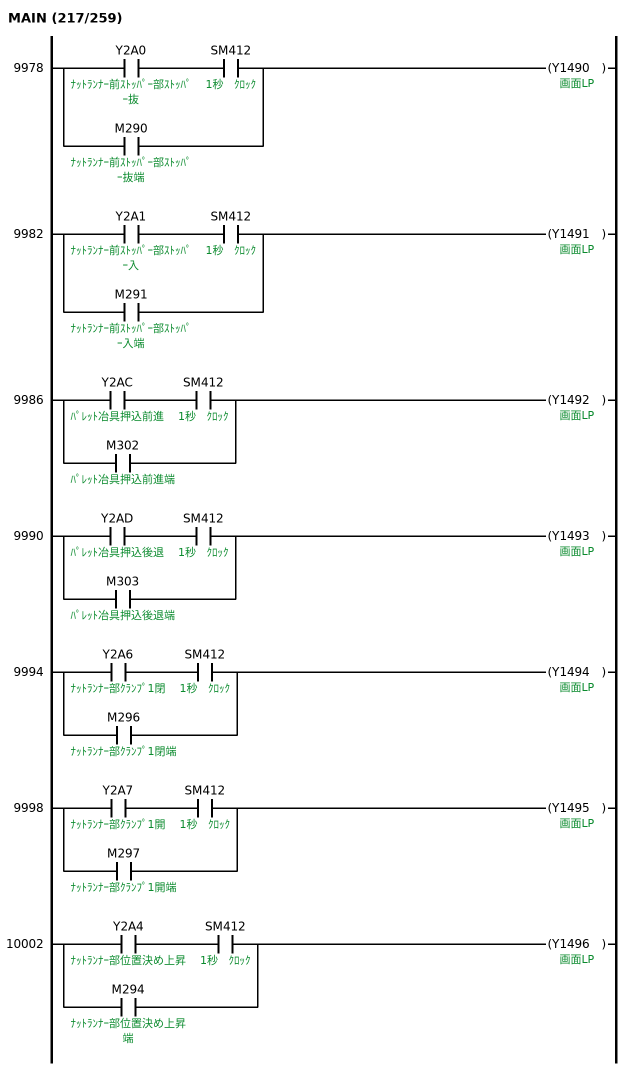
[picture p216: ladder of MAIN, rungs at steps 9978 to 10002]
9978  LD      Y2A0  ; ﾅｯﾄﾗﾝﾅｰ前ｽﾄｯﾊﾟｰ部ｽﾄｯﾊﾟｰ抜
      AND     SM412  ; 1秒   ｸﾛｯｸ
      OR      M290  ; ﾅｯﾄﾗﾝﾅｰ前ｽﾄｯﾊﾟｰ部ｽﾄｯﾊﾟｰ抜端
      OUT     Y1490  ; 画面LP
9982  LD      Y2A1  ; ﾅｯﾄﾗﾝﾅｰ前ｽﾄｯﾊﾟｰ部ｽﾄｯﾊﾟｰ入
      AND     SM412  ; 1秒   ｸﾛｯｸ
      OR      M291  ; ﾅｯﾄﾗﾝﾅｰ前ｽﾄｯﾊﾟｰ部ｽﾄｯﾊﾟｰ入端
      OUT     Y1491  ; 画面LP
9986  LD      Y2AC  ; ﾊﾟﾚｯﾄ冶具押込前進
      AND     SM412  ; 1秒   ｸﾛｯｸ
      OR      M302  ; ﾊﾟﾚｯﾄ冶具押込前進端
      OUT     Y1492  ; 画面LP
9990  LD      Y2AD  ; ﾊﾟﾚｯﾄ冶具押込後退
      AND     SM412  ; 1秒   ｸﾛｯｸ
      OR      M303  ; ﾊﾟﾚｯﾄ冶具押込後退端
      OUT     Y1493  ; 画面LP
9994  LD      Y2A6  ; ﾅｯﾄﾗﾝﾅｰ部ｸﾗﾝﾌﾟ1閉
      AND     SM412  ; 1秒   ｸﾛｯｸ
      OR      M296  ; ﾅｯﾄﾗﾝﾅｰ部ｸﾗﾝﾌﾟ1閉端
      OUT     Y1494  ; 画面LP
9998  LD      Y2A7  ; ﾅｯﾄﾗﾝﾅｰ部ｸﾗﾝﾌﾟ1開
      AND     SM412  ; 1秒   ｸﾛｯｸ
      OR      M297  ; ﾅｯﾄﾗﾝﾅｰ部ｸﾗﾝﾌﾟ1開端
      OUT     Y1495  ; 画面LP
10002 LD      Y2A4  ; ﾅｯﾄﾗﾝﾅｰ部位置決め上昇
      AND     SM412  ; 1秒   ｸﾛｯｸ
      OR      M294  ; ﾅｯﾄﾗﾝﾅｰ部位置決め上昇端
      OUT     Y1496  ; 画面LP
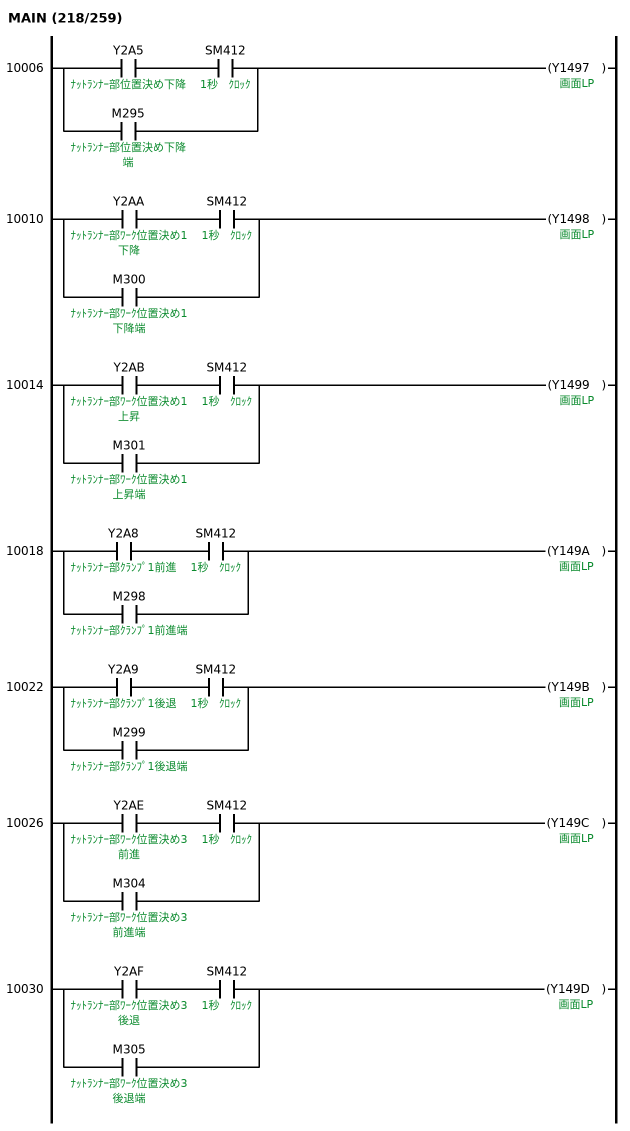
10006 LD      Y2A5  ; ﾅｯﾄﾗﾝﾅｰ部位置決め下降
      AND     SM412  ; 1秒   ｸﾛｯｸ
      OR      M295  ; ﾅｯﾄﾗﾝﾅｰ部位置決め下降端
      OUT     Y1497  ; 画面LP
10010 LD      Y2AA  ; ﾅｯﾄﾗﾝﾅｰ部ﾜｰｸ位置決め1下降
      AND     SM412  ; 1秒   ｸﾛｯｸ
      OR      M300  ; ﾅｯﾄﾗﾝﾅｰ部ﾜｰｸ位置決め1下降端
      OUT     Y1498  ; 画面LP
10014 LD      Y2AB  ; ﾅｯﾄﾗﾝﾅｰ部ﾜｰｸ位置決め1上昇
      AND     SM412  ; 1秒   ｸﾛｯｸ
      OR      M301  ; ﾅｯﾄﾗﾝﾅｰ部ﾜｰｸ位置決め1上昇端
      OUT     Y1499  ; 画面LP
10018 LD      Y2A8  ; ﾅｯﾄﾗﾝﾅｰ部ｸﾗﾝﾌﾟ1前進
      AND     SM412  ; 1秒   ｸﾛｯｸ
      OR      M298  ; ﾅｯﾄﾗﾝﾅｰ部ｸﾗﾝﾌﾟ1前進端
      OUT     Y149A  ; 画面LP
10022 LD      Y2A9  ; ﾅｯﾄﾗﾝﾅｰ部ｸﾗﾝﾌﾟ1後退
      AND     SM412  ; 1秒   ｸﾛｯｸ
      OR      M299  ; ﾅｯﾄﾗﾝﾅｰ部ｸﾗﾝﾌﾟ1後退端
      OUT     Y149B  ; 画面LP
10026 LD      Y2AE  ; ﾅｯﾄﾗﾝﾅｰ部ﾜｰｸ位置決め3前進
      AND     SM412  ; 1秒   ｸﾛｯｸ
      OR      M304  ; ﾅｯﾄﾗﾝﾅｰ部ﾜｰｸ位置決め3前進端
      OUT     Y149C  ; 画面LP
10030 LD      Y2AF  ; ﾅｯﾄﾗﾝﾅｰ部ﾜｰｸ位置決め3後退
      AND     SM412  ; 1秒   ｸﾛｯｸ
      OR      M305  ; ﾅｯﾄﾗﾝﾅｰ部ﾜｰｸ位置決め3後退端
      OUT     Y149D  ; 画面LP
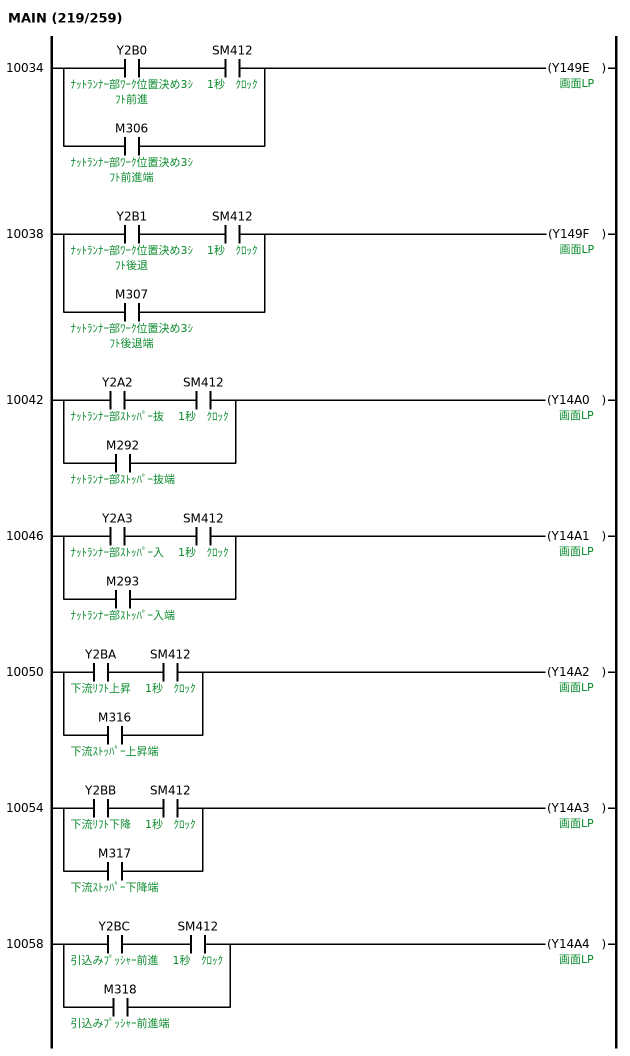
10034 LD      Y2B0  ; ﾅｯﾄﾗﾝﾅｰ部ﾜｰｸ位置決め3ｼﾌﾄ前進
      AND     SM412  ; 1秒   ｸﾛｯｸ
      OR      M306  ; ﾅｯﾄﾗﾝﾅｰ部ﾜｰｸ位置決め3ｼﾌﾄ前進端
      OUT     Y149E  ; 画面LP
10038 LD      Y2B1  ; ﾅｯﾄﾗﾝﾅｰ部ﾜｰｸ位置決め3ｼﾌﾄ後退
      AND     SM412  ; 1秒   ｸﾛｯｸ
      OR      M307  ; ﾅｯﾄﾗﾝﾅｰ部ﾜｰｸ位置決め3ｼﾌﾄ後退端
      OUT     Y149F  ; 画面LP
10042 LD      Y2A2  ; ﾅｯﾄﾗﾝﾅｰ部ｽﾄｯﾊﾟｰ抜
      AND     SM412  ; 1秒   ｸﾛｯｸ
      OR      M292  ; ﾅｯﾄﾗﾝﾅｰ部ｽﾄｯﾊﾟｰ抜端
      OUT     Y14A0  ; 画面LP
10046 LD      Y2A3  ; ﾅｯﾄﾗﾝﾅｰ部ｽﾄｯﾊﾟｰ入
      AND     SM412  ; 1秒   ｸﾛｯｸ
      OR      M293  ; ﾅｯﾄﾗﾝﾅｰ部ｽﾄｯﾊﾟｰ入端
      OUT     Y14A1  ; 画面LP
10050 LD      Y2BA  ; 下流ﾘﾌﾄ上昇
      AND     SM412  ; 1秒   ｸﾛｯｸ
      OR      M316  ; 下流ｽﾄｯﾊﾟｰ上昇端
      OUT     Y14A2  ; 画面LP
10054 LD      Y2BB  ; 下流ﾘﾌﾄ下降
      AND     SM412  ; 1秒   ｸﾛｯｸ
      OR      M317  ; 下流ｽﾄｯﾊﾟｰ下降端
      OUT     Y14A3  ; 画面LP
10058 LD      Y2BC  ; 引込みﾌﾟｯｼｬｰ前進
      AND     SM412  ; 1秒   ｸﾛｯｸ
      OR      M318  ; 引込みﾌﾟｯｼｬｰ前進端
      OUT     Y14A4  ; 画面LP
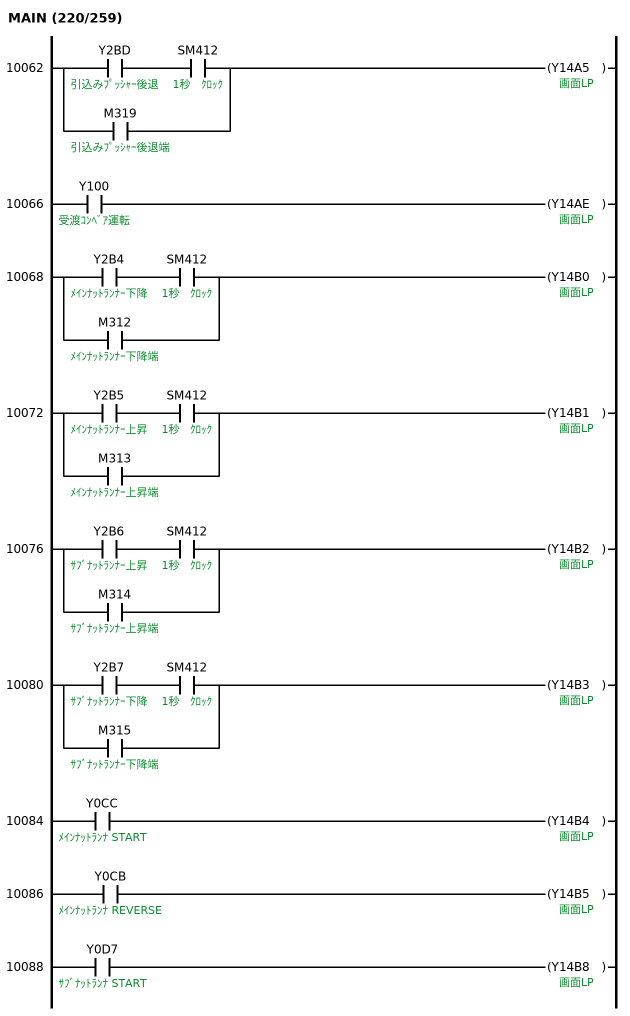
10062 LD      Y2BD  ; 引込みﾌﾟｯｼｬｰ後退
      AND     SM412  ; 1秒   ｸﾛｯｸ
      OR      M319  ; 引込みﾌﾟｯｼｬｰ後退端
      OUT     Y14A5  ; 画面LP
10066 LD      Y100  ; 受渡ｺﾝﾍﾞｱ運転
      OUT     Y14AE  ; 画面LP
10068 LD      Y2B4  ; ﾒｲﾝﾅｯﾄﾗﾝﾅｰ下降
      AND     SM412  ; 1秒   ｸﾛｯｸ
      OR      M312  ; ﾒｲﾝﾅｯﾄﾗﾝﾅｰ下降端
      OUT     Y14B0  ; 画面LP
10072 LD      Y2B5  ; ﾒｲﾝﾅｯﾄﾗﾝﾅｰ上昇
      AND     SM412  ; 1秒   ｸﾛｯｸ
      OR      M313  ; ﾒｲﾝﾅｯﾄﾗﾝﾅｰ上昇端
      OUT     Y14B1  ; 画面LP
10076 LD      Y2B6  ; ｻﾌﾞﾅｯﾄﾗﾝﾅｰ上昇
      AND     SM412  ; 1秒   ｸﾛｯｸ
      OR      M314  ; ｻﾌﾞﾅｯﾄﾗﾝﾅｰ上昇端
      OUT     Y14B2  ; 画面LP
10080 LD      Y2B7  ; ｻﾌﾞﾅｯﾄﾗﾝﾅｰ下降
      AND     SM412  ; 1秒   ｸﾛｯｸ
      OR      M315  ; ｻﾌﾞﾅｯﾄﾗﾝﾅｰ下降端
      OUT     Y14B3  ; 画面LP
10084 LD      Y0CC  ; ﾒｲﾝﾅｯﾄﾗﾝﾅ START
      OUT     Y14B4  ; 画面LP
10086 LD      Y0CB  ; ﾒｲﾝﾅｯﾄﾗﾝﾅ REVERSE
      OUT     Y14B5  ; 画面LP
10088 LD      Y0D7  ; ｻﾌﾞﾅｯﾄﾗﾝﾅ START
      OUT     Y14B8  ; 画面LP
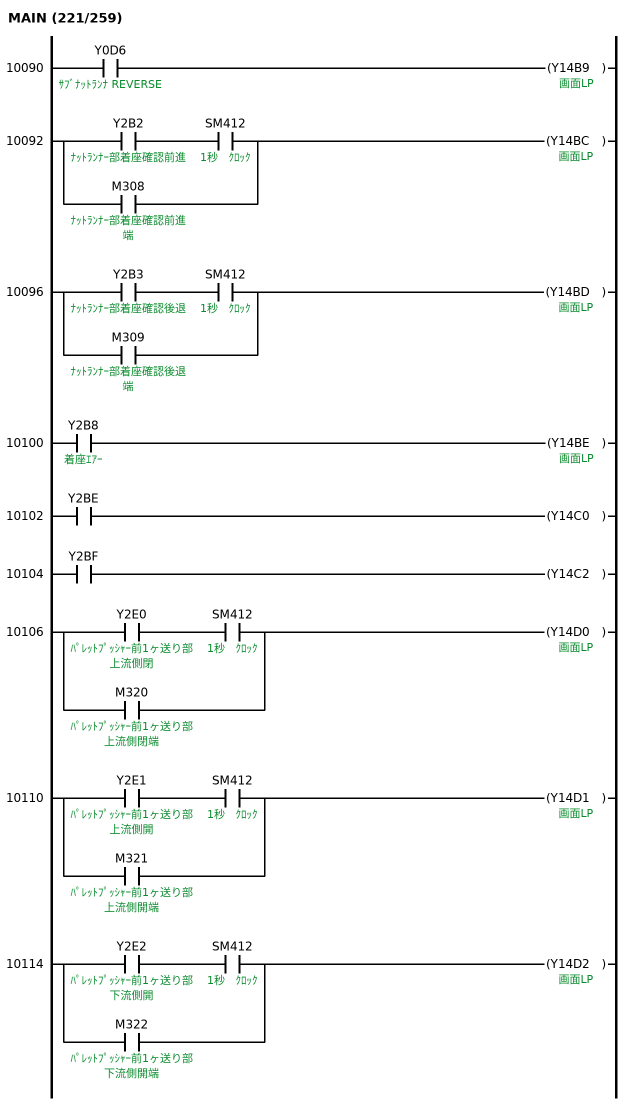
10090 LD      Y0D6  ; ｻﾌﾞﾅｯﾄﾗﾝﾅ REVERSE
      OUT     Y14B9  ; 画面LP
10092 LD      Y2B2  ; ﾅｯﾄﾗﾝﾅｰ部着座確認前進
      AND     SM412  ; 1秒   ｸﾛｯｸ
      OR      M308  ; ﾅｯﾄﾗﾝﾅｰ部着座確認前進端
      OUT     Y14BC  ; 画面LP
10096 LD      Y2B3  ; ﾅｯﾄﾗﾝﾅｰ部着座確認後退
      AND     SM412  ; 1秒   ｸﾛｯｸ
      OR      M309  ; ﾅｯﾄﾗﾝﾅｰ部着座確認後退端
      OUT     Y14BD  ; 画面LP
10100 LD      Y2B8  ; 着座ｴｱｰ
      OUT     Y14BE  ; 画面LP
10102 LD      Y2BE
      OUT     Y14C0
10104 LD      Y2BF
      OUT     Y14C2
10106 LD      Y2E0  ; ﾊﾟﾚｯﾄﾌﾟｯｼｬｰ前1ヶ送り部上流側閉
      AND     SM412  ; 1秒   ｸﾛｯｸ
      OR      M320  ; ﾊﾟﾚｯﾄﾌﾟｯｼｬｰ前1ヶ送り部上流側閉端
      OUT     Y14D0  ; 画面LP
10110 LD      Y2E1  ; ﾊﾟﾚｯﾄﾌﾟｯｼｬｰ前1ヶ送り部上流側開
      AND     SM412  ; 1秒   ｸﾛｯｸ
      OR      M321  ; ﾊﾟﾚｯﾄﾌﾟｯｼｬｰ前1ヶ送り部上流側開端
      OUT     Y14D1  ; 画面LP
10114 LD      Y2E2  ; ﾊﾟﾚｯﾄﾌﾟｯｼｬｰ前1ヶ送り部下流側開
      AND     SM412  ; 1秒   ｸﾛｯｸ
      OR      M322  ; ﾊﾟﾚｯﾄﾌﾟｯｼｬｰ前1ヶ送り部下流側開端
      OUT     Y14D2  ; 画面LP
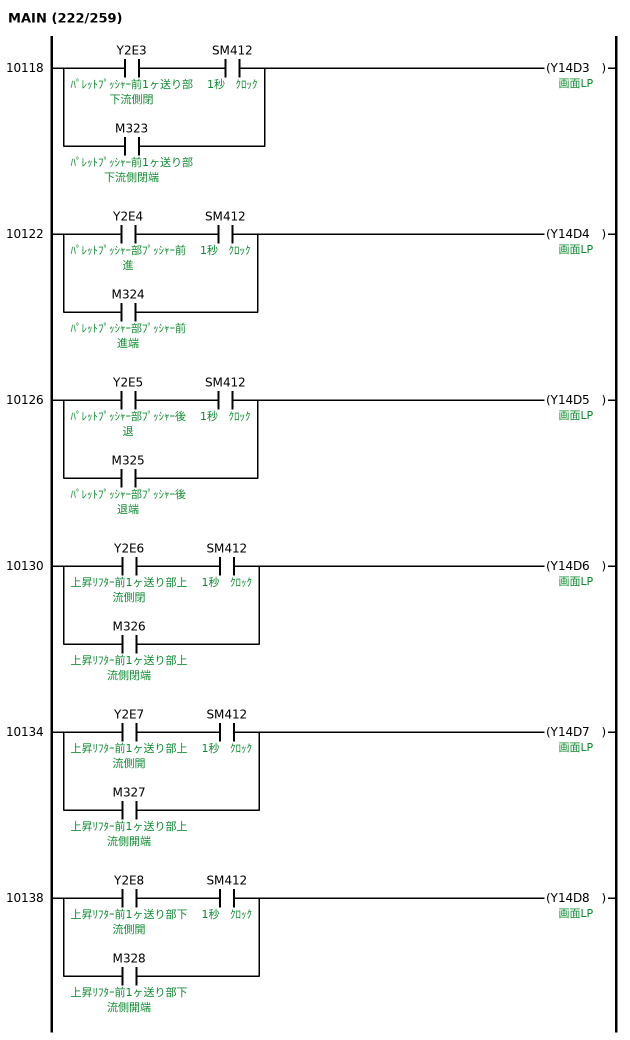
10118 LD      Y2E3  ; ﾊﾟﾚｯﾄﾌﾟｯｼｬｰ前1ヶ送り部下流側閉
      AND     SM412  ; 1秒   ｸﾛｯｸ
      OR      M323  ; ﾊﾟﾚｯﾄﾌﾟｯｼｬｰ前1ヶ送り部下流側閉端
      OUT     Y14D3  ; 画面LP
10122 LD      Y2E4  ; ﾊﾟﾚｯﾄﾌﾟｯｼｬｰ部ﾌﾟｯｼｬｰ前進
      AND     SM412  ; 1秒   ｸﾛｯｸ
      OR      M324  ; ﾊﾟﾚｯﾄﾌﾟｯｼｬｰ部ﾌﾟｯｼｬｰ前進端
      OUT     Y14D4  ; 画面LP
10126 LD      Y2E5  ; ﾊﾟﾚｯﾄﾌﾟｯｼｬｰ部ﾌﾟｯｼｬｰ後退
      AND     SM412  ; 1秒   ｸﾛｯｸ
      OR      M325  ; ﾊﾟﾚｯﾄﾌﾟｯｼｬｰ部ﾌﾟｯｼｬｰ後退端
      OUT     Y14D5  ; 画面LP
10130 LD      Y2E6  ; 上昇ﾘﾌﾀｰ前1ヶ送り部上流側閉
      AND     SM412  ; 1秒   ｸﾛｯｸ
      OR      M326  ; 上昇ﾘﾌﾀｰ前1ヶ送り部上流側閉端
      OUT     Y14D6  ; 画面LP
10134 LD      Y2E7  ; 上昇ﾘﾌﾀｰ前1ヶ送り部上流側開
      AND     SM412  ; 1秒   ｸﾛｯｸ
      OR      M327  ; 上昇ﾘﾌﾀｰ前1ヶ送り部上流側開端
      OUT     Y14D7  ; 画面LP
10138 LD      Y2E8  ; 上昇ﾘﾌﾀｰ前1ヶ送り部下流側開
      AND     SM412  ; 1秒   ｸﾛｯｸ
      OR      M328  ; 上昇ﾘﾌﾀｰ前1ヶ送り部下流側開端
      OUT     Y14D8  ; 画面LP
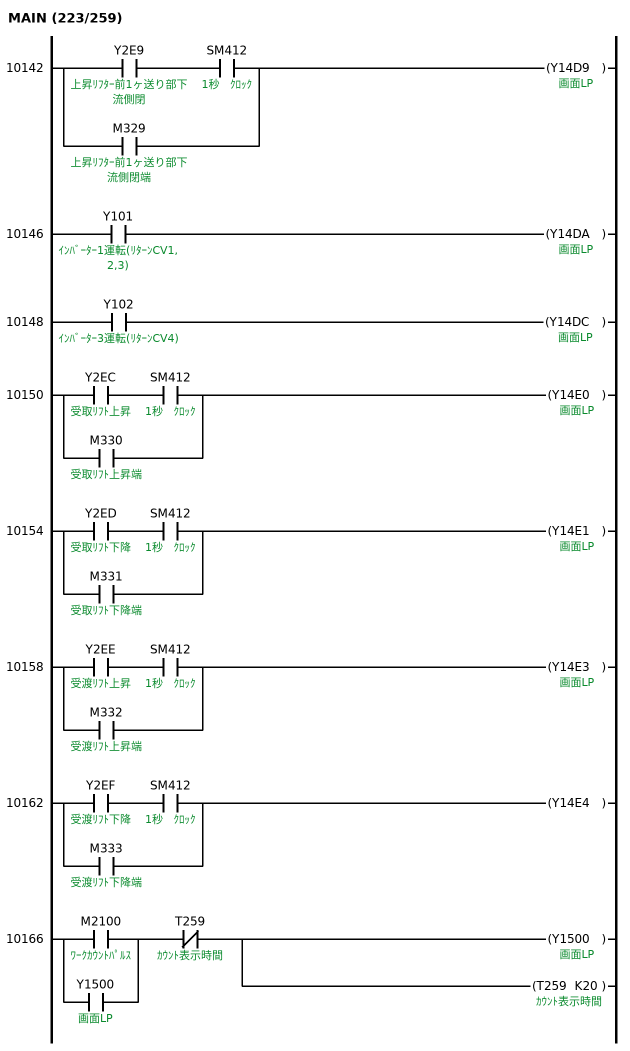
10142 LD      Y2E9  ; 上昇ﾘﾌﾀｰ前1ヶ送り部下流側閉
      AND     SM412  ; 1秒   ｸﾛｯｸ
      OR      M329  ; 上昇ﾘﾌﾀｰ前1ヶ送り部下流側閉端
      OUT     Y14D9  ; 画面LP
10146 LD      Y101  ; ｲﾝﾊﾞｰﾀｰ1運転(ﾘﾀｰﾝCV1,2,3)
      OUT     Y14DA  ; 画面LP
10148 LD      Y102  ; ｲﾝﾊﾞｰﾀｰ3運転(ﾘﾀｰﾝCV4)
      OUT     Y14DC  ; 画面LP
10150 LD      Y2EC  ; 受取ﾘﾌﾄ上昇
      AND     SM412  ; 1秒   ｸﾛｯｸ
      OR      M330  ; 受取ﾘﾌﾄ上昇端
      OUT     Y14E0  ; 画面LP
10154 LD      Y2ED  ; 受取ﾘﾌﾄ下降
      AND     SM412  ; 1秒   ｸﾛｯｸ
      OR      M331  ; 受取ﾘﾌﾄ下降端
      OUT     Y14E1  ; 画面LP
10158 LD      Y2EE  ; 受渡ﾘﾌﾄ上昇
      AND     SM412  ; 1秒   ｸﾛｯｸ
      OR      M332  ; 受渡ﾘﾌﾄ上昇端
      OUT     Y14E3  ; 画面LP
10162 LD      Y2EF  ; 受渡ﾘﾌﾄ下降
      AND     SM412  ; 1秒   ｸﾛｯｸ
      OR      M333  ; 受渡ﾘﾌﾄ下降端
      OUT     Y14E4
10166 LD      M2100  ; ﾜｰｸｶｳﾝﾄﾊﾟﾙｽ
      OR      Y1500  ; 画面LP
      ANI     T259  ; ｶｳﾝﾄ表示時間
      OUT     Y1500  ; 画面LP
      OUT     T259 K20  ; ｶｳﾝﾄ表示時間
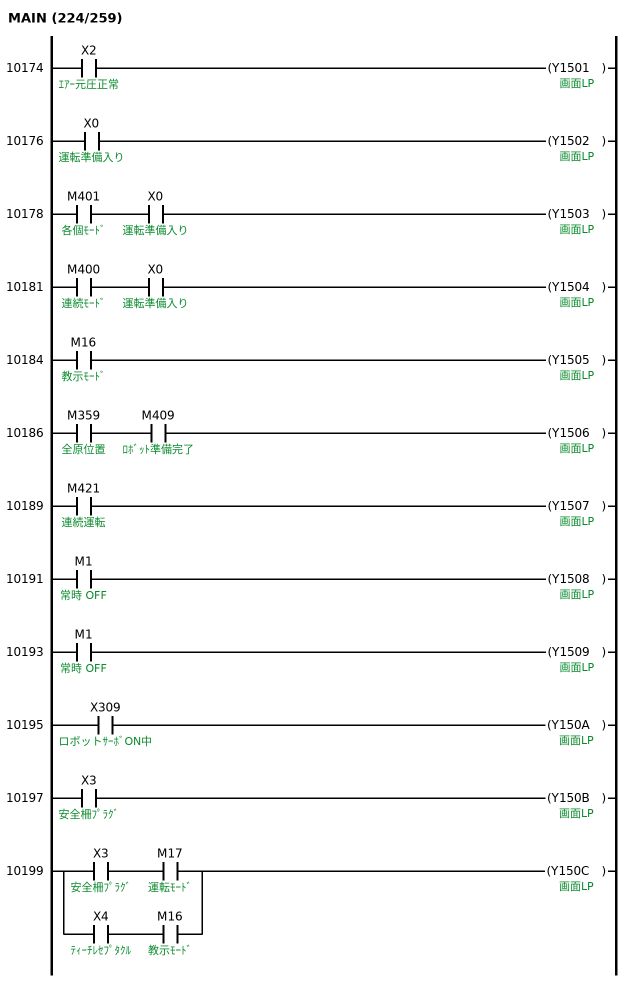
10174 LD      X2  ; ｴｱｰ元圧正常
      OUT     Y1501  ; 画面LP
10176 LD      X0  ; 運転準備入り
      OUT     Y1502  ; 画面LP
10178 LD      M401  ; 各個ﾓｰﾄﾞ
      AND     X0  ; 運転準備入り
      OUT     Y1503  ; 画面LP
10181 LD      M400  ; 連続ﾓｰﾄﾞ
      AND     X0  ; 運転準備入り
      OUT     Y1504  ; 画面LP
10184 LD      M16  ; 教示ﾓｰﾄﾞ
      OUT     Y1505  ; 画面LP
10186 LD      M359  ; 全原位置
      AND     M409  ; ﾛﾎﾞｯﾄ準備完了
      OUT     Y1506  ; 画面LP
10189 LD      M421  ; 連続運転
      OUT     Y1507  ; 画面LP
10191 LD      M1  ; 常時 OFF
      OUT     Y1508  ; 画面LP
10193 LD      M1  ; 常時 OFF
      OUT     Y1509  ; 画面LP
10195 LD      X309  ; ロボットｻｰﾎﾞON中
      OUT     Y150A  ; 画面LP
10197 LD      X3  ; 安全柵ﾌﾟﾗｸﾞ
      OUT     Y150B  ; 画面LP
10199 LD      X3  ; 安全柵ﾌﾟﾗｸﾞ
      AND     M17  ; 運転ﾓｰﾄﾞ
      LD      X4  ; ﾃｨｰﾁﾚｾﾌﾟﾀｸﾙ
      AND     M16  ; 教示ﾓｰﾄﾞ
      ORB
      OUT     Y150C  ; 画面LP
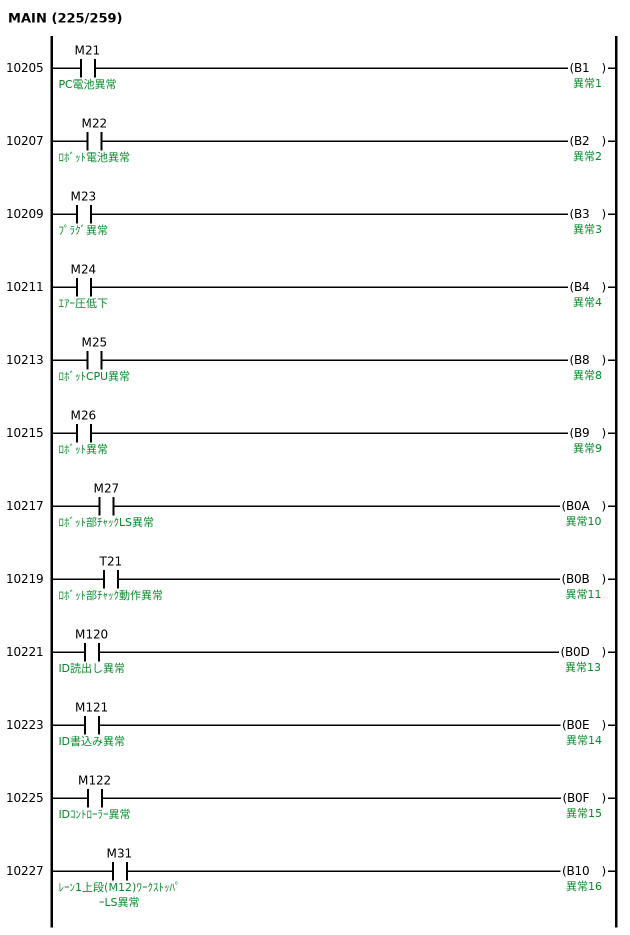
10205 LD      M21  ; PC電池異常
      OUT     B1  ; 異常1
10207 LD      M22  ; ﾛﾎﾞｯﾄ電池異常
      OUT     B2  ; 異常2
10209 LD      M23  ; ﾌﾟﾗｸﾞ異常
      OUT     B3  ; 異常3
10211 LD      M24  ; ｴｱｰ圧低下
      OUT     B4  ; 異常4
10213 LD      M25  ; ﾛﾎﾞｯﾄCPU異常
      OUT     B8  ; 異常8
10215 LD      M26  ; ﾛﾎﾞｯﾄ異常
      OUT     B9  ; 異常9
10217 LD      M27  ; ﾛﾎﾞｯﾄ部ﾁｬｯｸLS異常
      OUT     B0A  ; 異常10
10219 LD      T21  ; ﾛﾎﾞｯﾄ部ﾁｬｯｸ動作異常
      OUT     B0B  ; 異常11
10221 LD      M120  ; ID読出し異常
      OUT     B0D  ; 異常13
10223 LD      M121  ; ID書込み異常
      OUT     B0E  ; 異常14
10225 LD      M122  ; IDｺﾝﾄﾛｰﾗｰ異常
      OUT     B0F  ; 異常15
10227 LD      M31  ; ﾚｰﾝ1上段(M12)ﾜｰｸｽﾄｯﾊﾟｰLS異常
      OUT     B10  ; 異常16
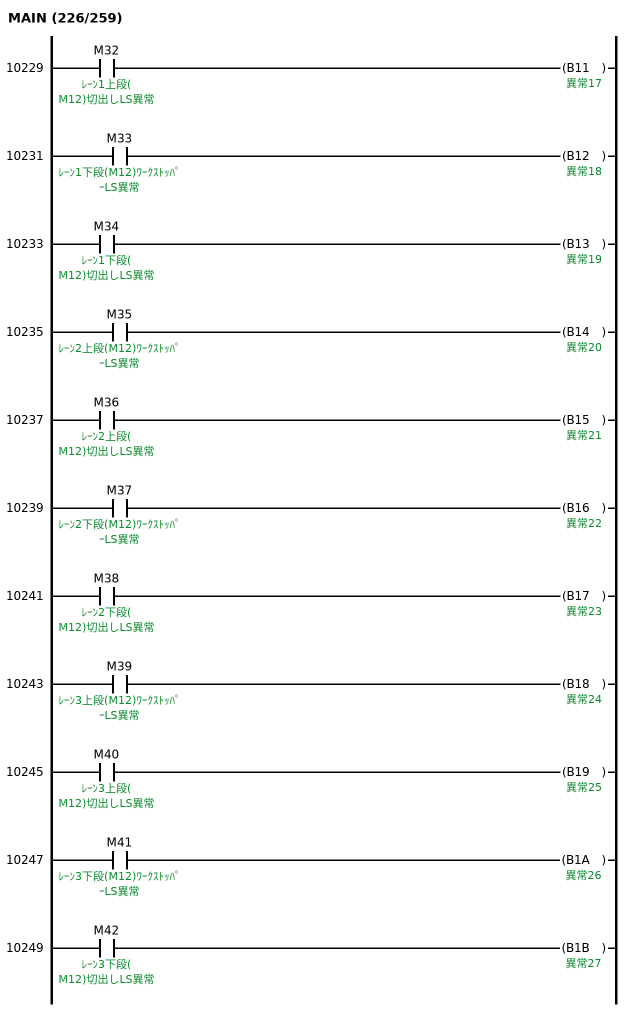
10229 LD      M32  ; ﾚｰﾝ1上段(M12)切出しLS異常
      OUT     B11  ; 異常17
10231 LD      M33  ; ﾚｰﾝ1下段(M12)ﾜｰｸｽﾄｯﾊﾟｰLS異常
      OUT     B12  ; 異常18
10233 LD      M34  ; ﾚｰﾝ1下段(M12)切出しLS異常
      OUT     B13  ; 異常19
10235 LD      M35  ; ﾚｰﾝ2上段(M12)ﾜｰｸｽﾄｯﾊﾟｰLS異常
      OUT     B14  ; 異常20
10237 LD      M36  ; ﾚｰﾝ2上段(M12)切出しLS異常
      OUT     B15  ; 異常21
10239 LD      M37  ; ﾚｰﾝ2下段(M12)ﾜｰｸｽﾄｯﾊﾟｰLS異常
      OUT     B16  ; 異常22
10241 LD      M38  ; ﾚｰﾝ2下段(M12)切出しLS異常
      OUT     B17  ; 異常23
10243 LD      M39  ; ﾚｰﾝ3上段(M12)ﾜｰｸｽﾄｯﾊﾟｰLS異常
      OUT     B18  ; 異常24
10245 LD      M40  ; ﾚｰﾝ3上段(M12)切出しLS異常
      OUT     B19  ; 異常25
10247 LD      M41  ; ﾚｰﾝ3下段(M12)ﾜｰｸｽﾄｯﾊﾟｰLS異常
      OUT     B1A  ; 異常26
10249 LD      M42  ; ﾚｰﾝ3下段(M12)切出しLS異常
      OUT     B1B  ; 異常27
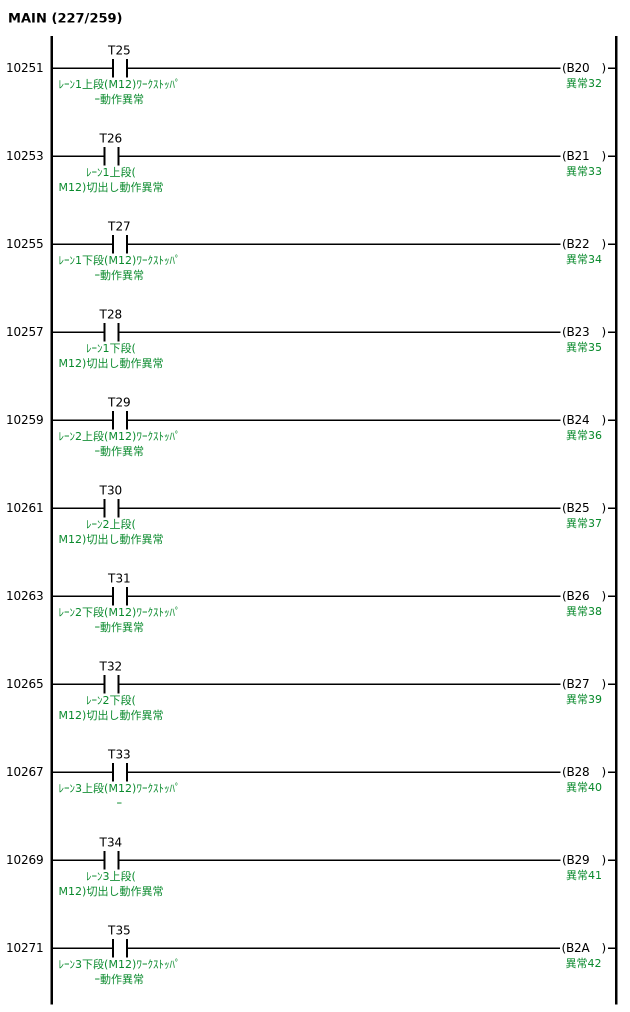
10251 LD      T25  ; ﾚｰﾝ1上段(M12)ﾜｰｸｽﾄｯﾊﾟｰ動作異常
      OUT     B20  ; 異常32
10253 LD      T26  ; ﾚｰﾝ1上段(M12)切出し動作異常
      OUT     B21  ; 異常33
10255 LD      T27  ; ﾚｰﾝ1下段(M12)ﾜｰｸｽﾄｯﾊﾟｰ動作異常
      OUT     B22  ; 異常34
10257 LD      T28  ; ﾚｰﾝ1下段(M12)切出し動作異常
      OUT     B23  ; 異常35
10259 LD      T29  ; ﾚｰﾝ2上段(M12)ﾜｰｸｽﾄｯﾊﾟｰ動作異常
      OUT     B24  ; 異常36
10261 LD      T30  ; ﾚｰﾝ2上段(M12)切出し動作異常
      OUT     B25  ; 異常37
10263 LD      T31  ; ﾚｰﾝ2下段(M12)ﾜｰｸｽﾄｯﾊﾟｰ動作異常
      OUT     B26  ; 異常38
10265 LD      T32  ; ﾚｰﾝ2下段(M12)切出し動作異常
      OUT     B27  ; 異常39
10267 LD      T33  ; ﾚｰﾝ3上段(M12)ﾜｰｸｽﾄｯﾊﾟｰ
      OUT     B28  ; 異常40
10269 LD      T34  ; ﾚｰﾝ3上段(M12)切出し動作異常
      OUT     B29  ; 異常41
10271 LD      T35  ; ﾚｰﾝ3下段(M12)ﾜｰｸｽﾄｯﾊﾟｰ動作異常
      OUT     B2A  ; 異常42
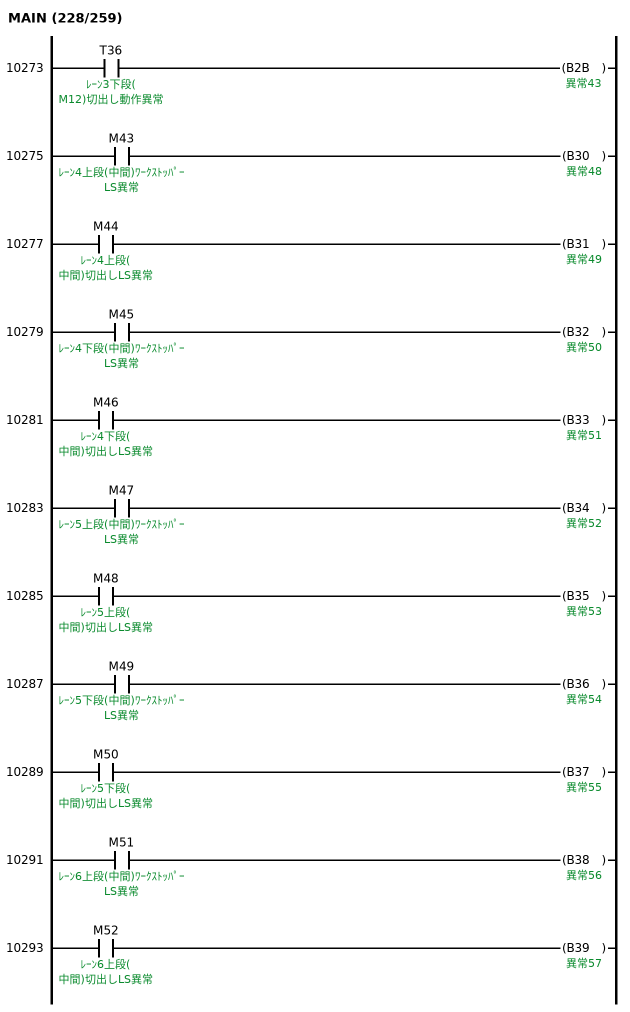
10273 LD      T36  ; ﾚｰﾝ3下段(M12)切出し動作異常
      OUT     B2B  ; 異常43
10275 LD      M43  ; ﾚｰﾝ4上段(中間)ﾜｰｸｽﾄｯﾊﾟｰLS異常
      OUT     B30  ; 異常48
10277 LD      M44  ; ﾚｰﾝ4上段(中間)切出しLS異常
      OUT     B31  ; 異常49
10279 LD      M45  ; ﾚｰﾝ4下段(中間)ﾜｰｸｽﾄｯﾊﾟｰLS異常
      OUT     B32  ; 異常50
10281 LD      M46  ; ﾚｰﾝ4下段(中間)切出しLS異常
      OUT     B33  ; 異常51
10283 LD      M47  ; ﾚｰﾝ5上段(中間)ﾜｰｸｽﾄｯﾊﾟｰLS異常
      OUT     B34  ; 異常52
10285 LD      M48  ; ﾚｰﾝ5上段(中間)切出しLS異常
      OUT     B35  ; 異常53
10287 LD      M49  ; ﾚｰﾝ5下段(中間)ﾜｰｸｽﾄｯﾊﾟｰLS異常
      OUT     B36  ; 異常54
10289 LD      M50  ; ﾚｰﾝ5下段(中間)切出しLS異常
      OUT     B37  ; 異常55
10291 LD      M51  ; ﾚｰﾝ6上段(中間)ﾜｰｸｽﾄｯﾊﾟｰLS異常
      OUT     B38  ; 異常56
10293 LD      M52  ; ﾚｰﾝ6上段(中間)切出しLS異常
      OUT     B39  ; 異常57
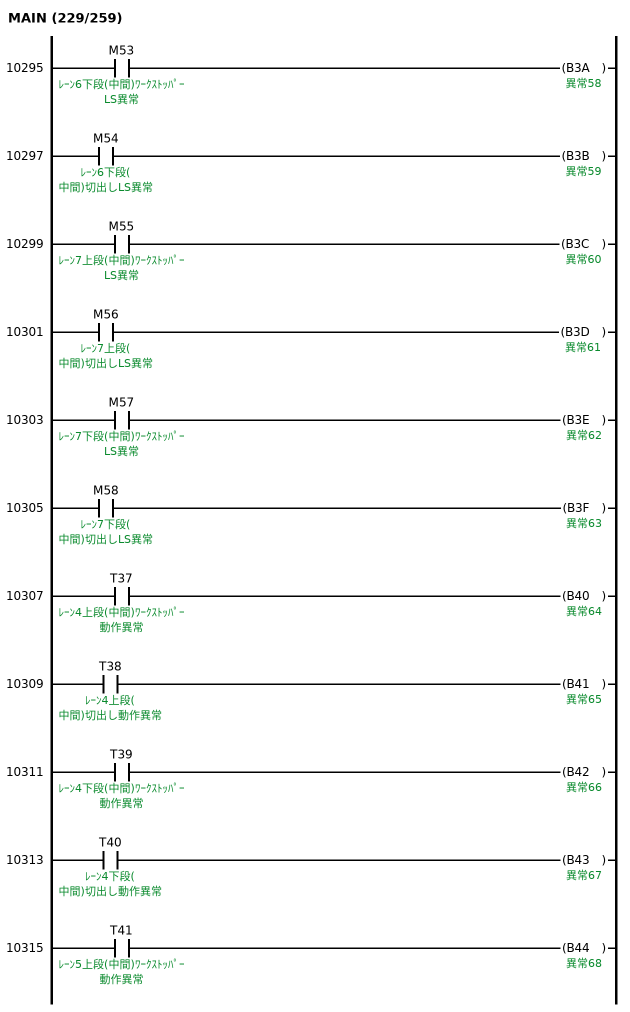
10295 LD      M53  ; ﾚｰﾝ6下段(中間)ﾜｰｸｽﾄｯﾊﾟｰLS異常
      OUT     B3A  ; 異常58
10297 LD      M54  ; ﾚｰﾝ6下段(中間)切出しLS異常
      OUT     B3B  ; 異常59
10299 LD      M55  ; ﾚｰﾝ7上段(中間)ﾜｰｸｽﾄｯﾊﾟｰLS異常
      OUT     B3C  ; 異常60
10301 LD      M56  ; ﾚｰﾝ7上段(中間)切出しLS異常
      OUT     B3D  ; 異常61
10303 LD      M57  ; ﾚｰﾝ7下段(中間)ﾜｰｸｽﾄｯﾊﾟｰLS異常
      OUT     B3E  ; 異常62
10305 LD      M58  ; ﾚｰﾝ7下段(中間)切出しLS異常
      OUT     B3F  ; 異常63
10307 LD      T37  ; ﾚｰﾝ4上段(中間)ﾜｰｸｽﾄｯﾊﾟｰ動作異常
      OUT     B40  ; 異常64
10309 LD      T38  ; ﾚｰﾝ4上段(中間)切出し動作異常
      OUT     B41  ; 異常65
10311 LD      T39  ; ﾚｰﾝ4下段(中間)ﾜｰｸｽﾄｯﾊﾟｰ動作異常
      OUT     B42  ; 異常66
10313 LD      T40  ; ﾚｰﾝ4下段(中間)切出し動作異常
      OUT     B43  ; 異常67
10315 LD      T41  ; ﾚｰﾝ5上段(中間)ﾜｰｸｽﾄｯﾊﾟｰ動作異常
      OUT     B44  ; 異常68
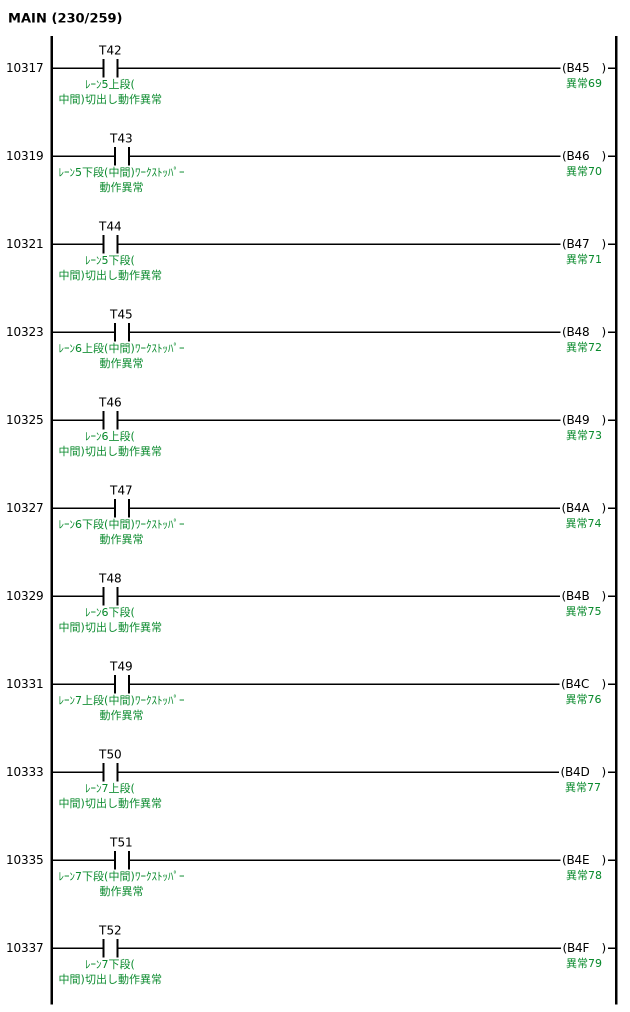
10317 LD      T42  ; ﾚｰﾝ5上段(中間)切出し動作異常
      OUT     B45  ; 異常69
10319 LD      T43  ; ﾚｰﾝ5下段(中間)ﾜｰｸｽﾄｯﾊﾟｰ動作異常
      OUT     B46  ; 異常70
10321 LD      T44  ; ﾚｰﾝ5下段(中間)切出し動作異常
      OUT     B47  ; 異常71
10323 LD      T45  ; ﾚｰﾝ6上段(中間)ﾜｰｸｽﾄｯﾊﾟｰ動作異常
      OUT     B48  ; 異常72
10325 LD      T46  ; ﾚｰﾝ6上段(中間)切出し動作異常
      OUT     B49  ; 異常73
10327 LD      T47  ; ﾚｰﾝ6下段(中間)ﾜｰｸｽﾄｯﾊﾟｰ動作異常
      OUT     B4A  ; 異常74
10329 LD      T48  ; ﾚｰﾝ6下段(中間)切出し動作異常
      OUT     B4B  ; 異常75
10331 LD      T49  ; ﾚｰﾝ7上段(中間)ﾜｰｸｽﾄｯﾊﾟｰ動作異常
      OUT     B4C  ; 異常76
10333 LD      T50  ; ﾚｰﾝ7上段(中間)切出し動作異常
      OUT     B4D  ; 異常77
10335 LD      T51  ; ﾚｰﾝ7下段(中間)ﾜｰｸｽﾄｯﾊﾟｰ動作異常
      OUT     B4E  ; 異常78
10337 LD      T52  ; ﾚｰﾝ7下段(中間)切出し動作異常
      OUT     B4F  ; 異常79
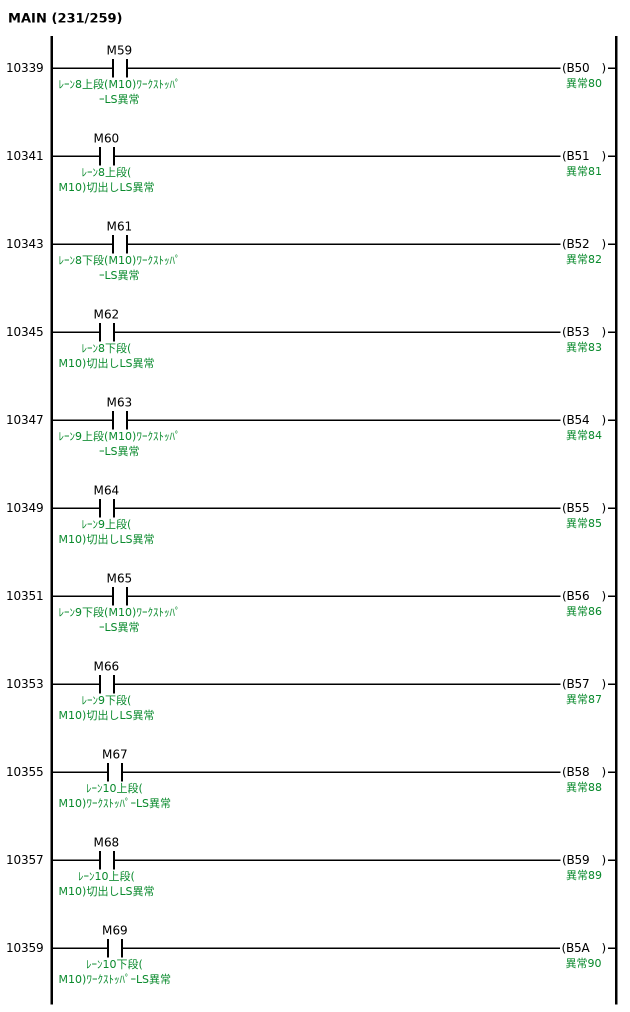
10339 LD      M59  ; ﾚｰﾝ8上段(M10)ﾜｰｸｽﾄｯﾊﾟｰLS異常
      OUT     B50  ; 異常80
10341 LD      M60  ; ﾚｰﾝ8上段(M10)切出しLS異常
      OUT     B51  ; 異常81
10343 LD      M61  ; ﾚｰﾝ8下段(M10)ﾜｰｸｽﾄｯﾊﾟｰLS異常
      OUT     B52  ; 異常82
10345 LD      M62  ; ﾚｰﾝ8下段(M10)切出しLS異常
      OUT     B53  ; 異常83
10347 LD      M63  ; ﾚｰﾝ9上段(M10)ﾜｰｸｽﾄｯﾊﾟｰLS異常
      OUT     B54  ; 異常84
10349 LD      M64  ; ﾚｰﾝ9上段(M10)切出しLS異常
      OUT     B55  ; 異常85
10351 LD      M65  ; ﾚｰﾝ9下段(M10)ﾜｰｸｽﾄｯﾊﾟｰLS異常
      OUT     B56  ; 異常86
10353 LD      M66  ; ﾚｰﾝ9下段(M10)切出しLS異常
      OUT     B57  ; 異常87
10355 LD      M67  ; ﾚｰﾝ10上段(M10)ﾜｰｸｽﾄｯﾊﾟｰLS異常
      OUT     B58  ; 異常88
10357 LD      M68  ; ﾚｰﾝ10上段(M10)切出しLS異常
      OUT     B59  ; 異常89
10359 LD      M69  ; ﾚｰﾝ10下段(M10)ﾜｰｸｽﾄｯﾊﾟｰLS異常
      OUT     B5A  ; 異常90
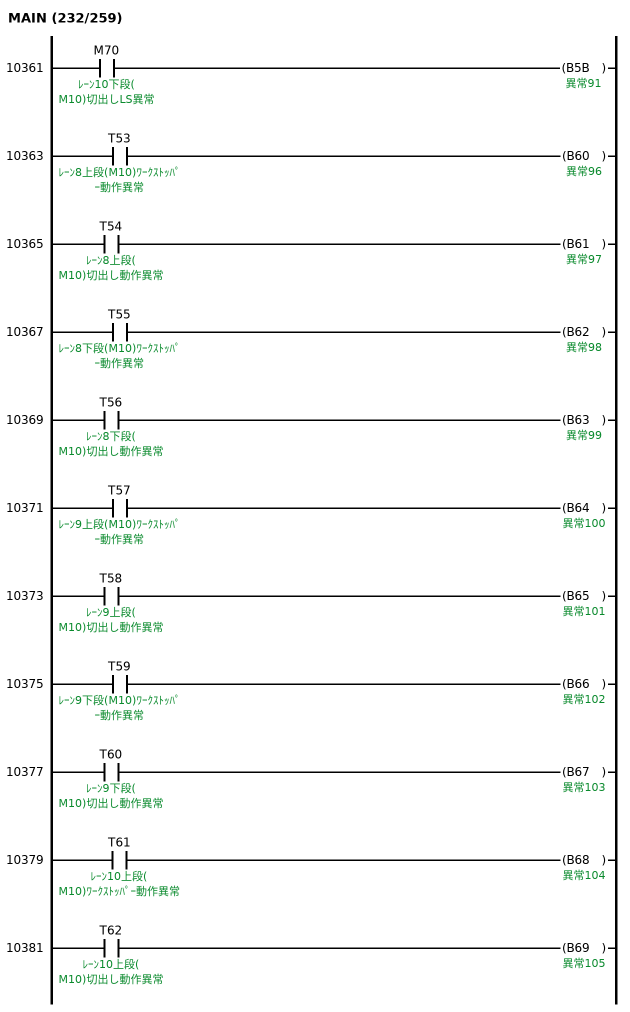
10361 LD      M70  ; ﾚｰﾝ10下段(M10)切出しLS異常
      OUT     B5B  ; 異常91
10363 LD      T53  ; ﾚｰﾝ8上段(M10)ﾜｰｸｽﾄｯﾊﾟｰ動作異常
      OUT     B60  ; 異常96
10365 LD      T54  ; ﾚｰﾝ8上段(M10)切出し動作異常
      OUT     B61  ; 異常97
10367 LD      T55  ; ﾚｰﾝ8下段(M10)ﾜｰｸｽﾄｯﾊﾟｰ動作異常
      OUT     B62  ; 異常98
10369 LD      T56  ; ﾚｰﾝ8下段(M10)切出し動作異常
      OUT     B63  ; 異常99
10371 LD      T57  ; ﾚｰﾝ9上段(M10)ﾜｰｸｽﾄｯﾊﾟｰ動作異常
      OUT     B64  ; 異常100
10373 LD      T58  ; ﾚｰﾝ9上段(M10)切出し動作異常
      OUT     B65  ; 異常101
10375 LD      T59  ; ﾚｰﾝ9下段(M10)ﾜｰｸｽﾄｯﾊﾟｰ動作異常
      OUT     B66  ; 異常102
10377 LD      T60  ; ﾚｰﾝ9下段(M10)切出し動作異常
      OUT     B67  ; 異常103
10379 LD      T61  ; ﾚｰﾝ10上段(M10)ﾜｰｸｽﾄｯﾊﾟｰ動作異常
      OUT     B68  ; 異常104
10381 LD      T62  ; ﾚｰﾝ10上段(M10)切出し動作異常
      OUT     B69  ; 異常105
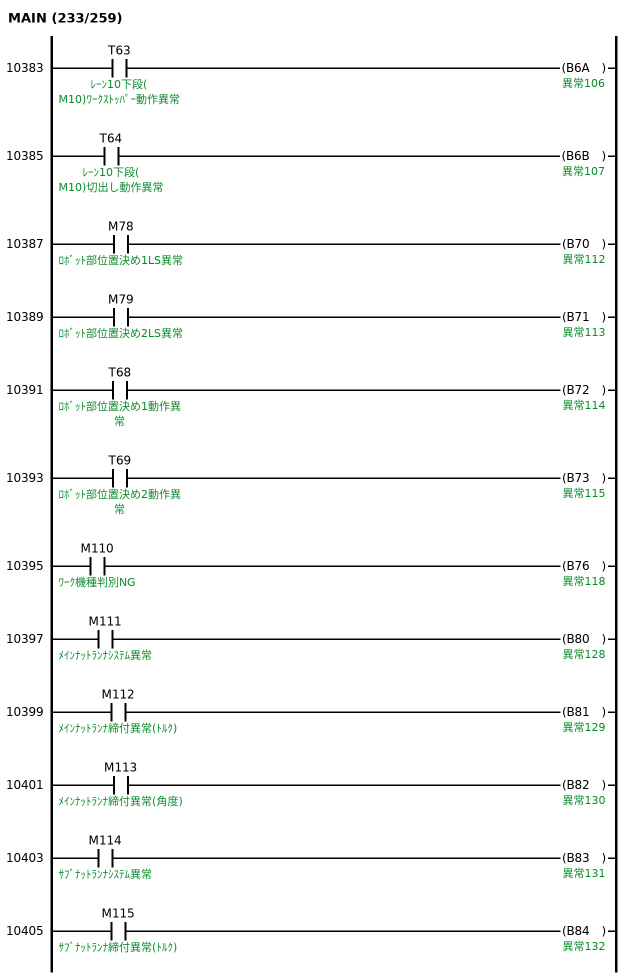
10383 LD      T63  ; ﾚｰﾝ10下段(M10)ﾜｰｸｽﾄｯﾊﾟｰ動作異常
      OUT     B6A  ; 異常106
10385 LD      T64  ; ﾚｰﾝ10下段(M10)切出し動作異常
      OUT     B6B  ; 異常107
10387 LD      M78  ; ﾛﾎﾞｯﾄ部位置決め1LS異常
      OUT     B70  ; 異常112
10389 LD      M79  ; ﾛﾎﾞｯﾄ部位置決め2LS異常
      OUT     B71  ; 異常113
10391 LD      T68  ; ﾛﾎﾞｯﾄ部位置決め1動作異常
      OUT     B72  ; 異常114
10393 LD      T69  ; ﾛﾎﾞｯﾄ部位置決め2動作異常
      OUT     B73  ; 異常115
10395 LD      M110  ; ﾜｰｸ機種判別NG
      OUT     B76  ; 異常118
10397 LD      M111  ; ﾒｲﾝﾅｯﾄﾗﾝﾅｼｽﾃﾑ異常
      OUT     B80  ; 異常128
10399 LD      M112  ; ﾒｲﾝﾅｯﾄﾗﾝﾅ締付異常(ﾄﾙｸ)
      OUT     B81  ; 異常129
10401 LD      M113  ; ﾒｲﾝﾅｯﾄﾗﾝﾅ締付異常(角度)
      OUT     B82  ; 異常130
10403 LD      M114  ; ｻﾌﾞﾅｯﾄﾗﾝﾅｼｽﾃﾑ異常
      OUT     B83  ; 異常131
10405 LD      M115  ; ｻﾌﾞﾅｯﾄﾗﾝﾅ締付異常(ﾄﾙｸ)
      OUT     B84  ; 異常132
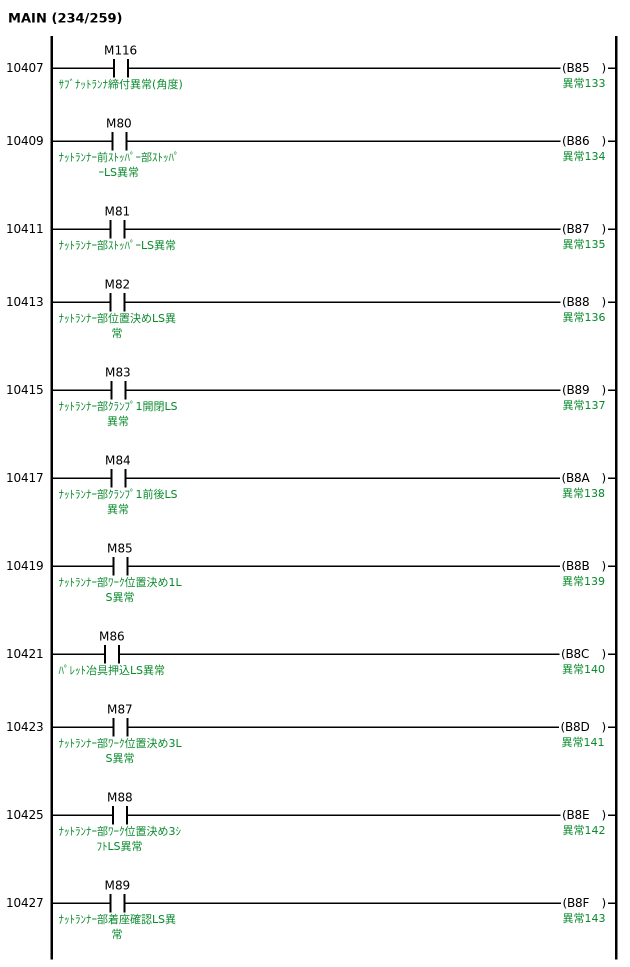
10407 LD      M116  ; ｻﾌﾞﾅｯﾄﾗﾝﾅ締付異常(角度)
      OUT     B85  ; 異常133
10409 LD      M80  ; ﾅｯﾄﾗﾝﾅｰ前ｽﾄｯﾊﾟｰ部ｽﾄｯﾊﾟｰLS異常
      OUT     B86  ; 異常134
10411 LD      M81  ; ﾅｯﾄﾗﾝﾅｰ部ｽﾄｯﾊﾟｰLS異常
      OUT     B87  ; 異常135
10413 LD      M82  ; ﾅｯﾄﾗﾝﾅｰ部位置決めLS異常
      OUT     B88  ; 異常136
10415 LD      M83  ; ﾅｯﾄﾗﾝﾅｰ部ｸﾗﾝﾌﾟ1開閉LS異常
      OUT     B89  ; 異常137
10417 LD      M84  ; ﾅｯﾄﾗﾝﾅｰ部ｸﾗﾝﾌﾟ1前後LS異常
      OUT     B8A  ; 異常138
10419 LD      M85  ; ﾅｯﾄﾗﾝﾅｰ部ﾜｰｸ位置決め1LS異常
      OUT     B8B  ; 異常139
10421 LD      M86  ; ﾊﾟﾚｯﾄ冶具押込LS異常
      OUT     B8C  ; 異常140
10423 LD      M87  ; ﾅｯﾄﾗﾝﾅｰ部ﾜｰｸ位置決め3LS異常
      OUT     B8D  ; 異常141
10425 LD      M88  ; ﾅｯﾄﾗﾝﾅｰ部ﾜｰｸ位置決め3ｼﾌﾄLS異常
      OUT     B8E  ; 異常142
10427 LD      M89  ; ﾅｯﾄﾗﾝﾅｰ部着座確認LS異常
      OUT     B8F  ; 異常143
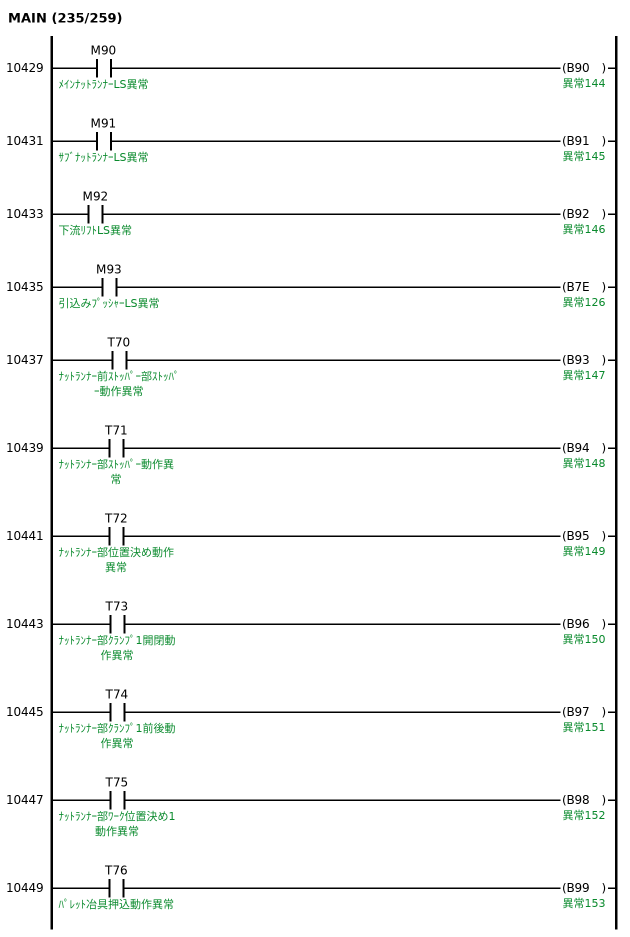
10429 LD      M90  ; ﾒｲﾝﾅｯﾄﾗﾝﾅｰLS異常
      OUT     B90  ; 異常144
10431 LD      M91  ; ｻﾌﾞﾅｯﾄﾗﾝﾅｰLS異常
      OUT     B91  ; 異常145
10433 LD      M92  ; 下流ﾘﾌﾄLS異常
      OUT     B92  ; 異常146
10435 LD      M93  ; 引込みﾌﾟｯｼｬｰLS異常
      OUT     B7E  ; 異常126
10437 LD      T70  ; ﾅｯﾄﾗﾝﾅｰ前ｽﾄｯﾊﾟｰ部ｽﾄｯﾊﾟｰ動作異常
      OUT     B93  ; 異常147
10439 LD      T71  ; ﾅｯﾄﾗﾝﾅｰ部ｽﾄｯﾊﾟｰ動作異常
      OUT     B94  ; 異常148
10441 LD      T72  ; ﾅｯﾄﾗﾝﾅｰ部位置決め動作異常
      OUT     B95  ; 異常149
10443 LD      T73  ; ﾅｯﾄﾗﾝﾅｰ部ｸﾗﾝﾌﾟ1開閉動作異常
      OUT     B96  ; 異常150
10445 LD      T74  ; ﾅｯﾄﾗﾝﾅｰ部ｸﾗﾝﾌﾟ1前後動作異常
      OUT     B97  ; 異常151
10447 LD      T75  ; ﾅｯﾄﾗﾝﾅｰ部ﾜｰｸ位置決め1動作異常
      OUT     B98  ; 異常152
10449 LD      T76  ; ﾊﾟﾚｯﾄ冶具押込動作異常
      OUT     B99  ; 異常153
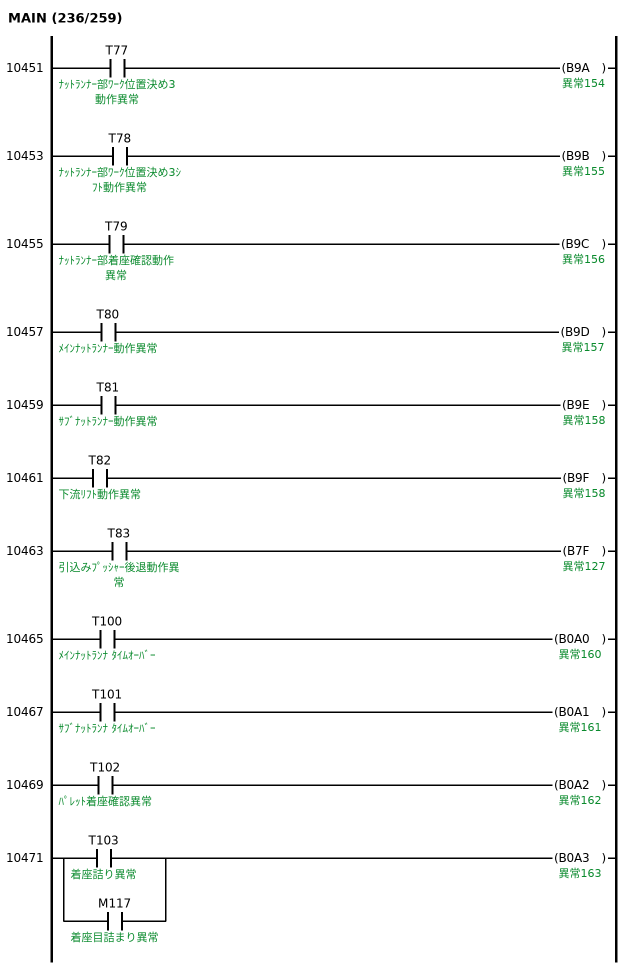
10451 LD      T77  ; ﾅｯﾄﾗﾝﾅｰ部ﾜｰｸ位置決め3動作異常
      OUT     B9A  ; 異常154
10453 LD      T78  ; ﾅｯﾄﾗﾝﾅｰ部ﾜｰｸ位置決め3ｼﾌﾄ動作異常
      OUT     B9B  ; 異常155
10455 LD      T79  ; ﾅｯﾄﾗﾝﾅｰ部着座確認動作異常
      OUT     B9C  ; 異常156
10457 LD      T80  ; ﾒｲﾝﾅｯﾄﾗﾝﾅｰ動作異常
      OUT     B9D  ; 異常157
10459 LD      T81  ; ｻﾌﾞﾅｯﾄﾗﾝﾅｰ動作異常
      OUT     B9E  ; 異常158
10461 LD      T82  ; 下流ﾘﾌﾄ動作異常
      OUT     B9F  ; 異常158
10463 LD      T83  ; 引込みﾌﾟｯｼｬｰ後退動作異常
      OUT     B7F  ; 異常127
10465 LD      T100  ; ﾒｲﾝﾅｯﾄﾗﾝﾅ ﾀｲﾑｵｰﾊﾞｰ
      OUT     B0A0  ; 異常160
10467 LD      T101  ; ｻﾌﾞﾅｯﾄﾗﾝﾅ ﾀｲﾑｵｰﾊﾞｰ
      OUT     B0A1  ; 異常161
10469 LD      T102  ; ﾊﾟﾚｯﾄ着座確認異常
      OUT     B0A2  ; 異常162
10471 LD      T103  ; 着座詰り異常
      OR      M117  ; 着座目詰まり異常
      OUT     B0A3  ; 異常163
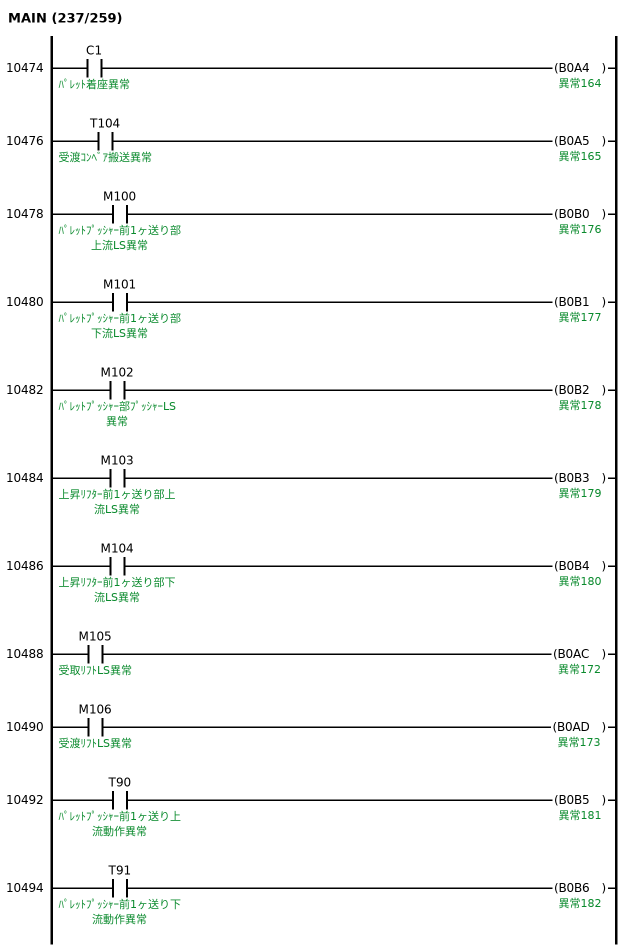
10474 LD      C1  ; ﾊﾟﾚｯﾄ着座異常
      OUT     B0A4  ; 異常164
10476 LD      T104  ; 受渡ｺﾝﾍﾞｱ搬送異常
      OUT     B0A5  ; 異常165
10478 LD      M100  ; ﾊﾟﾚｯﾄﾌﾟｯｼｬｰ前1ヶ送り部上流LS異常
      OUT     B0B0  ; 異常176
10480 LD      M101  ; ﾊﾟﾚｯﾄﾌﾟｯｼｬｰ前1ヶ送り部下流LS異常
      OUT     B0B1  ; 異常177
10482 LD      M102  ; ﾊﾟﾚｯﾄﾌﾟｯｼｬｰ部ﾌﾟｯｼｬｰLS異常
      OUT     B0B2  ; 異常178
10484 LD      M103  ; 上昇ﾘﾌﾀｰ前1ヶ送り部上流LS異常
      OUT     B0B3  ; 異常179
10486 LD      M104  ; 上昇ﾘﾌﾀｰ前1ヶ送り部下流LS異常
      OUT     B0B4  ; 異常180
10488 LD      M105  ; 受取ﾘﾌﾄLS異常
      OUT     B0AC  ; 異常172
10490 LD      M106  ; 受渡ﾘﾌﾄLS異常
      OUT     B0AD  ; 異常173
10492 LD      T90  ; ﾊﾟﾚｯﾄﾌﾟｯｼｬｰ前1ヶ送り上流動作異常
      OUT     B0B5  ; 異常181
10494 LD      T91  ; ﾊﾟﾚｯﾄﾌﾟｯｼｬｰ前1ヶ送り下流動作異常
      OUT     B0B6  ; 異常182
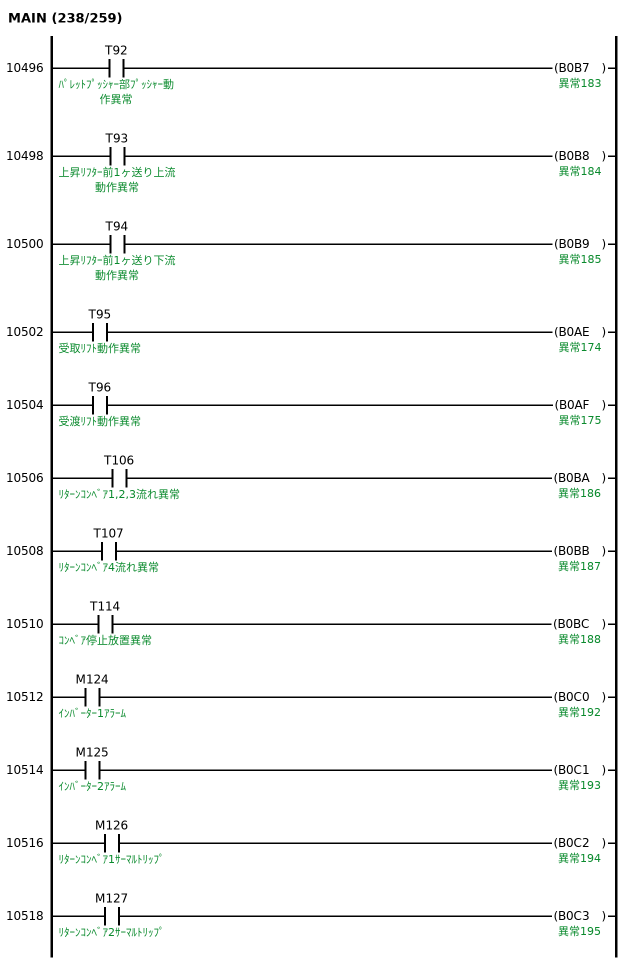
10496 LD      T92  ; ﾊﾟﾚｯﾄﾌﾟｯｼｬｰ部ﾌﾟｯｼｬｰ動作異常
      OUT     B0B7  ; 異常183
10498 LD      T93  ; 上昇ﾘﾌﾀｰ前1ヶ送り上流動作異常
      OUT     B0B8  ; 異常184
10500 LD      T94  ; 上昇ﾘﾌﾀｰ前1ヶ送り下流動作異常
      OUT     B0B9  ; 異常185
10502 LD      T95  ; 受取ﾘﾌﾄ動作異常
      OUT     B0AE  ; 異常174
10504 LD      T96  ; 受渡ﾘﾌﾄ動作異常
      OUT     B0AF  ; 異常175
10506 LD      T106  ; ﾘﾀｰﾝｺﾝﾍﾞｱ1,2,3流れ異常
      OUT     B0BA  ; 異常186
10508 LD      T107  ; ﾘﾀｰﾝｺﾝﾍﾞｱ4流れ異常
      OUT     B0BB  ; 異常187
10510 LD      T114  ; ｺﾝﾍﾞｱ停止放置異常
      OUT     B0BC  ; 異常188
10512 LD      M124  ; ｲﾝﾊﾞｰﾀｰ1ｱﾗｰﾑ
      OUT     B0C0  ; 異常192
10514 LD      M125  ; ｲﾝﾊﾞｰﾀｰ2ｱﾗｰﾑ
      OUT     B0C1  ; 異常193
10516 LD      M126  ; ﾘﾀｰﾝｺﾝﾍﾞｱ1ｻｰﾏﾙﾄﾘｯﾌﾟ
      OUT     B0C2  ; 異常194
10518 LD      M127  ; ﾘﾀｰﾝｺﾝﾍﾞｱ2ｻｰﾏﾙﾄﾘｯﾌﾟ
      OUT     B0C3  ; 異常195
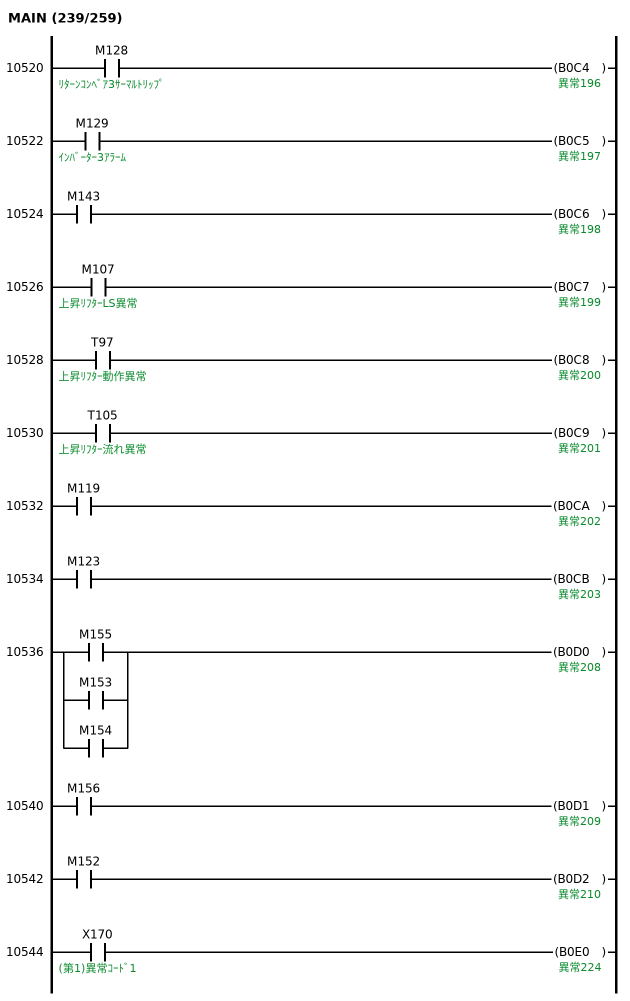
10520 LD      M128  ; ﾘﾀｰﾝｺﾝﾍﾞｱ3ｻｰﾏﾙﾄﾘｯﾌﾟ
      OUT     B0C4  ; 異常196
10522 LD      M129  ; ｲﾝﾊﾞｰﾀｰ3ｱﾗｰﾑ
      OUT     B0C5  ; 異常197
10524 LD      M143
      OUT     B0C6  ; 異常198
10526 LD      M107  ; 上昇ﾘﾌﾀｰLS異常
      OUT     B0C7  ; 異常199
10528 LD      T97  ; 上昇ﾘﾌﾀｰ動作異常
      OUT     B0C8  ; 異常200
10530 LD      T105  ; 上昇ﾘﾌﾀｰ流れ異常
      OUT     B0C9  ; 異常201
10532 LD      M119
      OUT     B0CA  ; 異常202
10534 LD      M123
      OUT     B0CB  ; 異常203
10536 LD      M155
      OR      M153
      OR      M154
      OUT     B0D0  ; 異常208
10540 LD      M156
      OUT     B0D1  ; 異常209
10542 LD      M152
      OUT     B0D2  ; 異常210
10544 LD      X170  ; (第1)異常ｺｰﾄﾞ1
      OUT     B0E0  ; 異常224
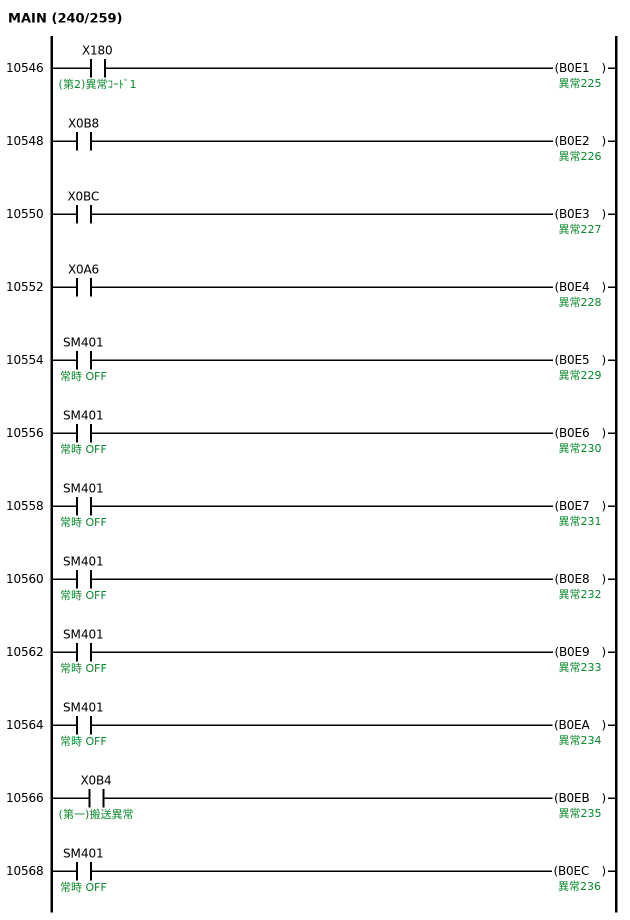
10546 LD      X180  ; (第2)異常ｺｰﾄﾞ1
      OUT     B0E1  ; 異常225
10548 LD      X0B8
      OUT     B0E2  ; 異常226
10550 LD      X0BC
      OUT     B0E3  ; 異常227
10552 LD      X0A6
      OUT     B0E4  ; 異常228
10554 LD      SM401  ; 常時 OFF
      OUT     B0E5  ; 異常229
10556 LD      SM401  ; 常時 OFF
      OUT     B0E6  ; 異常230
10558 LD      SM401  ; 常時 OFF
      OUT     B0E7  ; 異常231
10560 LD      SM401  ; 常時 OFF
      OUT     B0E8  ; 異常232
10562 LD      SM401  ; 常時 OFF
      OUT     B0E9  ; 異常233
10564 LD      SM401  ; 常時 OFF
      OUT     B0EA  ; 異常234
10566 LD      X0B4  ; (第一)搬送異常
      OUT     B0EB  ; 異常235
10568 LD      SM401  ; 常時 OFF
      OUT     B0EC  ; 異常236
